// TwinCAT 3 PLC project nn_inference
// ProgramVersion: 3.1.4024.0
// libraries:
//   Real-Time Neural Network Inference, * (ISW)
//   Tc2_Standard, * (Beckhoff Automation GmbH)
//   Tc2_System, * (Beckhoff Automation GmbH)
//   Tc2_Utilities, * (Beckhoff Automation GmbH)
//   Tc3_Module, * (Beckhoff Automation GmbH)
// project tree:
//   DUTs/ Dense_v1_Layers.TcDUT, Dense_v1_LayerWeights.TcDUT
//   / PlcTask.TcTTO
//   POUs/ FB_Dense_v1.TcPOU, MAIN.TcPOU
// real-time tasks:
//   TASK PlcTask: cycle T#10ms, priority 20, ADS port 350

CONFIGURATION nn_inference
    RESOURCE PLC ON TwinCAT3
        TASK PlcTask(INTERVAL := T#10ms, PRIORITY := 20);
        PROGRAM MAIN WITH PlcTask : MAIN;
    END_RESOURCE
END_CONFIGURATION

// ---- DUTs/Dense_v1_Layers.TcDUT

TYPE Dense_v1_Layers:
STRUCT
    num_layers : UINT := 5;
    weights : Dense_v1_LayerWeights;
    layers : ARRAY[0..4] OF Layer :=[
    (num_neurons := 5),
    (num_neurons := 100, activation := act_type.relu, pointer_weight:= ADR(weights.HiddenLayers1_weight),pointer_bias:= ADR(weights.HiddenLayers1_bias)),
    (num_neurons := 100, activation := act_type.relu, pointer_weight:= ADR(weights.HiddenLayers2_weight),pointer_bias:= ADR(weights.HiddenLayers2_bias)),
    (num_neurons := 100, activation := act_type.relu, pointer_weight:= ADR(weights.HiddenLayers3_weight),pointer_bias:= ADR(weights.HiddenLayers3_bias)),
    (num_neurons := 1, activation := act_type.linear, pointer_weight:= ADR(weights.OutputLayer_weight),pointer_bias:= ADR(weights.OutputLayer_bias))];
    layer_output : ARRAY[0..99] OF LREAL;
    layer_input : ARRAY[0..99] OF LREAL;
    
END_STRUCT
END_TYPE

// ---- DUTs/Dense_v1_LayerWeights.TcDUT

TYPE Dense_v1_LayerWeights:
STRUCT
    normalization_mean : ARRAY[0..0] OF LREAL;
    normalization_std : ARRAY[0..0] OF LREAL;
    HiddenLayers1_weight : ARRAY[0..99,0..4] OF LREAL;
    HiddenLayers1_bias : ARRAY[0..99] OF LREAL;
    HiddenLayers2_weight : ARRAY[0..99,0..99] OF LREAL;
    HiddenLayers2_bias : ARRAY[0..99] OF LREAL;
    HiddenLayers3_weight : ARRAY[0..99,0..99] OF LREAL;
    HiddenLayers3_bias : ARRAY[0..99] OF LREAL;
    OutputLayer_weight : ARRAY[0..0,0..99] OF LREAL;
    OutputLayer_bias : ARRAY[0..0] OF LREAL;
    denormalization_mean : ARRAY[0..0] OF LREAL;
    denormalization_std : ARRAY[0..0] OF LREAL;
    hash_sha_256 : ARRAY[0..3] OF LREAL;
END_STRUCT
END_TYPE

// ---- POUs/MAIN.TcPOU
PROGRAM MAIN
VAR
	input : ARRAY[0..4] OF LREAL := [1,1,1,1,1];
	out : ARRAY[0..0] OF LREAL;
	FB_nn : FB_Dense_v1;
END_VAR

FB_nn(pointer_input := ADR(input),pointer_output:=ADR(out));

END_PROGRAM

// ---- POUs/FB_Dense_v1.TcPOU

FUNCTION_BLOCK FB_Dense_v1
VAR_INPUT
	pointer_input: POINTER TO LREAL;
	pointer_output : POINTER TO LREAL;
	
END_VAR
VAR	
  i : UINT;
  flag_AreWeightsLoaded : BOOL := FALSE;
  flag_AreWeightsChecked : BOOL := FALSE;
  load_weights : FB_LoadWeights;
  filePath : T_MaxString := 'c:\Users\Administrator\Documents\git-projekte\keras2plc\examples\Python\test_ST_files\Dense_v1_weights.dat';
  nn : Dense_v1_Layers;
  hash_sha_256_twincat : ARRAY[0..3] OF LREAL;
  compare_res : DINT := 99;
END_VAR


IF NOT flag_AreWeightsLoaded THEN
		load_weights(execute := TRUE,filePath := filePath,ReadAdr := ADR(nn.weights), ReadLen :=  SIZEOF(nn.weights));
		IF NOT load_weights.busy THEN 
			flag_AreWeightsLoaded := TRUE;
		END_IF
ELSIF NOT flag_AreWeightsChecked THEN
	F_GenerateHashValue(hashMode:=E_HashMode.HASH_SHA256,pData := ADR(nn.weights),nData := SIZEOF(nn.weights)-32,pHash := ADR(hash_sha_256_twincat),nHash:=32);
	compare_res := MEMCMp(pBuf1 := ADR(hash_sha_256_twincat),ADR(nn.weights.hash_sha_256),32);
	IF compare_res = 0 THEN
		flag_AreWeightsChecked := TRUE;
	END_IF
ELSE
	MEMCPY(destAddr:=ADR(nn.layer_input),srcAddr:=pointer_input,n:=SIZEOF(LREAL)*nn.layers[0].num_neurons);

    
   // forward inference
	FOR i := 0 TO nn.num_layers-2 DO
		F_ForwardPropagation(	layer_pre	:= 	nn.layers[i],
								layer_next	:=	nn.layers[i+1],
								pointer_in 	:=	ADR(nn.layer_input),
								pointer_out	:=	ADR(nn.layer_output)	);
		MEMCPY(destAddr:=ADR(nn.layer_input),srcAddr:=ADR(nn.layer_output),n:=SIZEOF(LREAL)*nn.layers[i+1].num_neurons);
	END_FOR
	MEMCPY(destAddr:=pointer_output,srcAddr:=ADR(nn.layer_output),n:=SIZEOF(LREAL)*nn.layers[SIZEOF(nn.layers)/SIZEOF(nn.layers[0])-1].num_neurons);
    
    // output denormalization
    F_NormalizationLayer(pointer_input := pointer_output,pointer_mean := ADR(nn.weights.denormalization_mean),
    pointer_std := ADR(nn.weights.denormalization_std),invert := TRUE, num_neurons := nn.layers[SIZEOF(nn.layers)/SIZEOF(nn.layers[0])-1].num_neurons);    
END_IF

END_FUNCTION_BLOCK
